# EPICS autosave request: ADApp/Db/NDFileNexus_settings.req
$(P)$(R)TemplateFilePath
$(P)$(R)TemplateFileName
